TEXTLIST ISS_Object
  1 = 'C'
  2 = 'Y'
  3 = 'M'
  4 = 'K'
  5 = 'LC'
  6 = 'LM'
  7 = 'Prime'
  8 = 'W'
  9 = 'FUSH'
   = ''
END_TEXTLIST

(* stored: Version 1.1.0.1, ProductVersion 3.1.4024.11
   TextList ISS_Object: Id {e4b316b1-2344-4ff5-8e49-97a2acca8460} *)
